// SIMATIC S7-200 project (STEP 7-Micro/WIN), CPU 221 REL 01.10

ORGANIZATION_BLOCK MAIN:OB1
TITLE=PROGRAM COMMENTS
VAR
I0.0:?;	//  start
END_VAR
BEGIN
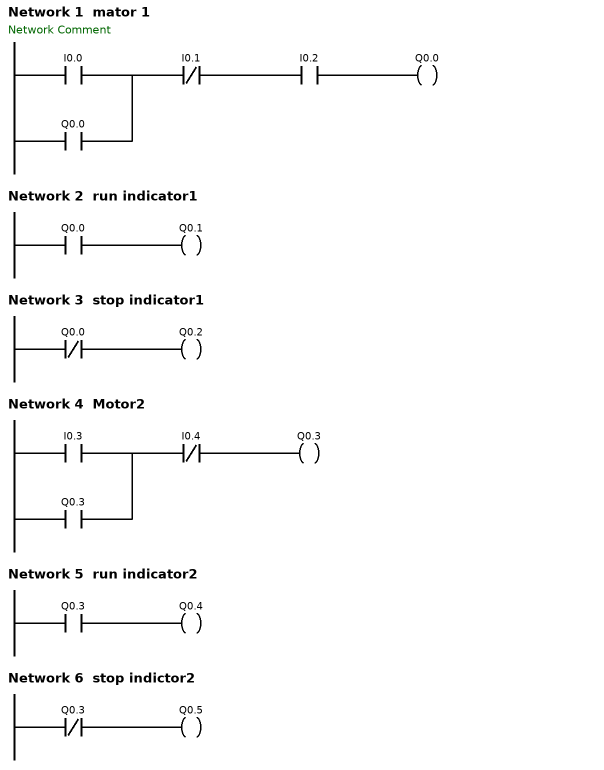
Network 1 // mator 1
// Network Comment
LD     I0.0
O      Q0.0
AN     I0.1
A      I0.2
=      Q0.0
Network 2 // run indicator1
LD     Q0.0
=      Q0.1
Network 3 // stop indicator1
LDN    Q0.0
=      Q0.2
Network 4 // Motor2
LD     I0.3
O      Q0.3
AN     I0.4
=      Q0.3
Network 5 // run indicator2
LD     Q0.3
=      Q0.4
Network 6 // stop indictor2
LDN    Q0.3
=      Q0.5
END_ORGANIZATION_BLOCK
